{attribute 'GeneratedUsingTerminal: EL3102--0000'}
{attribute addProperty BoxType "EL3102--0000"}
{attribute addProperty Id "StatusAT %I*BYTE1ValueAT %I*INT2"}
{attribute addProperty CRC "1966713395"}
{attribute addProperty Size "3"}
TYPE Channel_7539AA33 EXTENDS InputBase_8311D824 :
STRUCT
	{attribute addProperty Name "Status"}
	Status AT %I* : BYTE;
	{attribute addProperty Name "Value"}
	Value AT %I* : INT;
END_STRUCT
END_TYPE

(* stored: Version 1.2.0.0, ProductVersion 3.1.4024.9
   DUT Channel_7539AA33: Id {17e81538-e999-48f5-b22a-72b96a53a6e7} *)
